PROGRAM C08_PulseGenerator
VAR
	fbPulse05s					: FB_SquareWave;
	fbPulse1s						: FB_SquareWave;
	fbPulse2s						: FB_SquareWave;
	fbPulse5s						: FB_SquareWave;
	fbPulse10s					: FB_SquareWave;
END_VAR

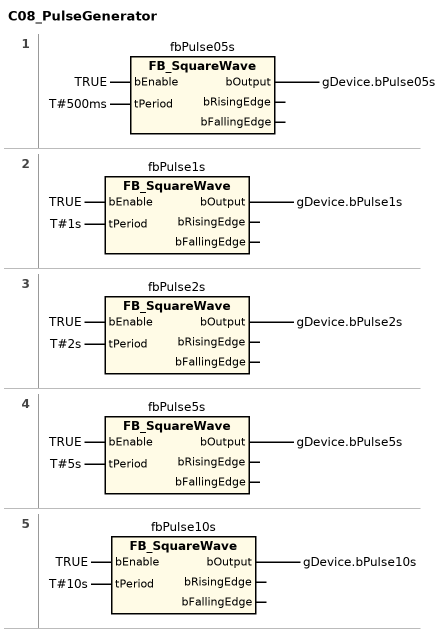
// NETWORK 1
fbPulse05s(bEnable := TRUE, tPeriod := T#500ms); // FB_SquareWave
gDevice.bPulse05s := fbPulse05s.bOutput;

// NETWORK 2
fbPulse1s(bEnable := TRUE, tPeriod := T#1s); // FB_SquareWave
gDevice.bPulse1s := fbPulse1s.bOutput;

// NETWORK 3
fbPulse2s(bEnable := TRUE, tPeriod := T#2s); // FB_SquareWave
gDevice.bPulse2s := fbPulse2s.bOutput;

// NETWORK 4
fbPulse5s(bEnable := TRUE, tPeriod := T#5s); // FB_SquareWave
gDevice.bPulse5s := fbPulse5s.bOutput;

// NETWORK 5
fbPulse10s(bEnable := TRUE, tPeriod := T#10s); // FB_SquareWave
gDevice.bPulse10s := fbPulse10s.bOutput;

END_PROGRAM

(* stored: Version 1.1.0.1
   POU C08_PulseGenerator: Id {82d07bad-b2de-417f-947b-e75d2d6a3d24}, SpecialFunc None *)
